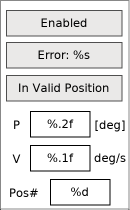
VISUALIZATION vAxisMainParamsDisplay  // 130x210
VAR_IN_OUT
	fbAxis	: FB_ServoAxis;
	fbTableControl :FB_TableControl;
END_VAR
    RoundedRectangle (0,0 129x257)
    Rectangle (30,111 60x26), "%.2f", text variable: fbAxis.McReadActualPosition.Axis.NcToPlc.ModuloActPos
    Label (93,112 34x26), "[deg]"
    Label (4,112 25x26), "P"
    Label (4,142 25x26)
    Rectangle (30,145 60x26), "%.1f", text variable: fbAxis.McReadActualVelocity.ActualVelocity, colour toggle: fbAxis.IsMoving
    Label (88,145 44x26), "deg/s"
    Label (4,146 25x26), "V"
    Rectangle (6,42 116x26), "Error: %s", text variable: TO_STRING(fbAxis.nActEvent), colour toggle: fbAxis.IsErrorActive
    Rectangle (6,10 116x26), "Enabled", colour toggle: fbAxis.Enabled
    Rectangle (6,213 116x26), "Details"
        OnMouseDown: execute { fbTableControl.stHMI.iDialogNumber := 100; }
    Label (-5,180 58x26), "Pos#"
    Rectangle (50,179 60x26), "%d", text variable: fbAxis.iCurrentPositionNumber, colour toggle: fbAxis.IsMoving
    Rectangle (6,75 116x26), "In Valid Position", colour toggle: fbAxis.bPositionValid
END_VISUALIZATION

(* stored: Version 1.1.0.1, ProductVersion 3.1.4024.15
   Visu vAxisMainParamsDisplay: Id {5564688d-a8af-4a2b-8e1a-268667f3c819} *)
